{attribute 'qualified_only'}
VAR_GLOBAL

	g_stProcessData : sProcessData;

	//Cycle Counter
	g_iCounter : INT := 0;
	
	//Control Button
	g_bStart : BOOL := FALSE;
    g_bStop  : BOOL := TRUE;
    g_bReset : BOOL := FALSE;
	g_bExit  : BOOL := FALSE;
END_VAR

(* stored: Version 1.1.0.1, ProductVersion 3.1.4024.15
   GVL GVL: Id {679680a8-c0b5-4f39-bc4f-3e6e594b9367} *)
